FUNCTION_BLOCK ABSTRACT CyclicComponent EXTENDS Component IMPLEMENTS I_Cyclic
VAR
	RegisteredAsCyclicResult : RegistrationResult;
END_VAR

METHOD ABSTRACT CyclicLogic
END_METHOD

METHOD DeregisterWithParent
VAR_INPUT
	Parent : I_ContainComponents;
END_VAR
Parent.DeregisterComponent(THIS^);
Parent.DeregisterCyclic(THIS^);
END_METHOD

METHOD RegisterWithParent
VAR_INPUT
	Parent : I_ContainComponents;
END_VAR
RegisteredAsComponentResult := Parent.RegisterComponent(THIS^);
RegisteredAsCyclicResult := Parent.RegisterCyclic(THIS^);
END_METHOD

END_FUNCTION_BLOCK

(* stored: Version 1.1.0.1, ProductVersion 3.1.4026.18
   POU CyclicComponent: Id {b2391d7a-f629-4dac-b0d6-c1bfe2964c84}, SpecialFunc None
   Method CyclicLogic: Id {e5abf98f-c2f8-44a5-a44b-6de6071ca988}
   Method DeregisterWithParent: Id {0ae9503f-d100-416f-9b08-0992249eb176}
   Method RegisterWithParent: Id {cbbbdde3-bad0-41d7-80fd-7b4457cdaea6} *)
